PROGRAM CurrentBPUpdate
VAR
    {attribute 'pytmc' := '
        pv: @(PREFIX)K:Rate
        link: IOC:BSY0:MP01:BYKIKS_RATE
        field: EGU RateEnum
    '}
    fbBYKIK_Rate : FB_LREALFromEPICS := (
        iMaximumValidSeverity := 2);


    {attribute 'pytmc' := '
        pv: @(PREFIX)
    '}
    fbEPICS_KRate : FB_RateFromEPICS;

    {attribute 'pytmc' := '
        pv: @(PREFIX)L:BC
        link: SIOC:SYS0:MP03:SC_SXR_BC
        field: EGU BCEnum
    '}
    fbMPS_BeamClass : FB_LREALFromEPICS := (
        iMaximumValidSeverity := 2);

        {attribute 'pytmc' := '
        pv: @(PREFIX)
    '}
    fbEPICSKBeamClass : FB_BeamClassFromEPICS;

    {attribute 'pytmc' := '
        pv: @(PREFIX)K:Mode
        link: SIOC:FEES:MP01:FACMODE_RBV
    '}
    fbSXR_MachineMode : FB_LREALFromEPICS := (
        iMaximumValidSeverity := 2);

    {attribute 'pytmc' := '
        pv: @(PREFIX)
    '}
    fbEPICSLMachineMode : FB_MachineModeFromEPICS;

    {attribute 'pytmc' := '
        pv: @(PREFIX)PE
    '}
    fbKPhotonEnergy : FB_KPhotonEnergy;

    // Photon energy for the masses
    {attribute 'TcLinkTo' := 'TIIB[plc-kfe-gatt]^IO Outputs^rPhotonEnergy'}
    {attribute 'TcLinkTo' := 'TIIB[plc-rix-mot]^IO Outputs^rPhotonEnergy'}
    {attribute 'TcLinkTo' := 'TIIB[plc-rix-optics]^IO Outputs^rPhotonEnergy'}
    q_rPhotonEnergy AT %Q* : REAL;


    // Stoppers

    {attribute 'TcLinkTo' := '
                .i_StopperInLS:=TIIB[PPS Stoppers 1]^Channel 1^ST3K4 IN;
                .i_StopperOutLS:=TIIB[PPS Stoppers 1]^Channel 2^ST3K4 OUT;
                .q_StopperIN_Relay:=TIIB[PMPS_Premp]^Channel 12^ST3K4 RELAY IN;
                                '}
    st3k4Watcher : FB_KStopper(
        PMPS.K_Stopper.ST3K4,
        'ST3K4');

   {attribute 'TcLinkTo' := '
                .i_StopperInLS:=TIIB[PPS Stoppers 1]^Channel 3^ST1K2 IN;
                .i_StopperOutLS:=TIIB[PPS Stoppers 1]^Channel 4^ST1K2 OUT;
                .q_StopperIN_Relay:=TIIB[PMPS_Premp]^Channel 14^ST1K2 RELAY IN;
                                '}
    st1k2Watcher : FB_KStopper(
        PMPS.K_Stopper.ST1K2,
        'ST1K2');

    {attribute 'TcLinkTo' := '
                .i_StopperInLS:=TIIB[PPS Stoppers 1]^Channel 5^ST1K3 IN;
                .i_StopperOutLS:=TIIB[PPS Stoppers 1]^Channel 6^ST1K3 OUT;
                .q_StopperIN_Relay:=TIIB[PMPS_Premp]^Channel 7^ST1K3 RELAY IN;
                                '}
    st1k3Watcher : FB_KStopper(
        PMPS.K_Stopper.ST1K3,
        'ST1K3');

    // MR1K1 Veto
    ////////////////////////
          {attribute 'TcLinkTo' := 'TIIB[plc-rix-optics]^IO Inputs^MR1K1_Y_ENC'}
        i_MR1K1_ENC AT %I* : UDINT; // MR1K1 encoder from the rix optics system
        cMR1K1_IN_UpperLimit : UDINT := 33411000;
        cMR1K1_IN_LowerLimit : UDINT := 31911000;
        cMR1K1_OUT_UpperLimit : UDINT := 14173400;
        {attribute 'TcLinkTo' := 'TIIB[PMPS_Premp]^Channel 13^MR1K1 IN'}
        q_MR1K1_VETO AT %Q* : BOOL; // Signal to accel. MPS that MR1K1 is in
        fbMR1K1VetoDevice : FB_KVetoDevice(
            eVetoDeviceIN := K_Stopper.MR1K1_IN,
            eVetoDeviceOUT := K_Stopper.MR1K1_OUT,
            sVetoDeviceName := 'MR1K1');




    // ST4K4 Photon Terminator Veto
    {attribute 'TcLinkTo' := '
                .i_StopperInLS:=TIIB[plc-tmo-mot]^IO Inputs^bST4K4_IN;
                .i_StopperOutLS:=TIIB[plc-tmo-mot]^IO Inputs^bST4K4_OUT;
     '}
    st4k4Watcher : FB_KStopper(
        PMPS.K_Stopper.ST4K4,
        'ST4K4');


     // MR1K3 Veto
    ////////////////////////
          {attribute 'TcLinkTo' := 'TIIB[plc-txi-optics]^IO Inputs^MR1K3_Y_ENC'}
        i_MR1K3_ENC AT %I* : ULINT; // MR1K3 encoder from the txi k optics optics system
        cMR1K3_IN_UpperLimit : UDINT := 108500000 + 10000000;
        cMR1K3_IN_LowerLimit : UDINT := 108500000 - 10000000 ;
        cMR1K3_OUT_UpperLimit : UDINT := 8900000 + 100000;

        q_MR1K3_VETO AT %Q* : BOOL; // Signal to accel. MPS that MR1K3 is in
        fbMR1K3VetoDevice : FB_KVetoDevice(
            eVetoDeviceIN := K_Stopper.MR1K3_IN,
            eVetoDeviceOUT := K_Stopper.MR1K3_OUT,
            sVetoDeviceName := 'MR1K3');

    // MR2K3 Veto
    ////////////////////////
          {attribute 'TcLinkTo' := 'TIIB[plc-txi-optics]^IO Inputs^MR2K3_Y_ENC'}
        i_MR2K3_ENC AT %I* : ULINT; // MR2K3 encoder from the txi k optics system
        cMR2K3_IN_UpperLimit : UDINT := 105650000 + 10000000;
        cMR2K3_IN_LowerLimit : UDINT := 105650000 - 10000000 ;
        cMR2K3_OUT_UpperLimit : UDINT := 10000000;

        q_MR2K3_VETO AT %Q* : BOOL; // Signal to accel. MPS that MR2K3 is in
        fbMR2K3VetoDevice : FB_KVetoDevice(
            eVetoDeviceIN := K_Stopper.MR2K3_IN,
            eVetoDeviceOUT := K_Stopper.MR2K3_OUT,
            sVetoDeviceName := 'MR2K3');


    // ST1K4Veto
    // ST1K4 Test Photon stopper Veto in the FEE right before ST3K4 stopper
    st1k4Watcher :   FB_KVetoDevice(
            eVetoDeviceIN := K_Stopper.ST1K4,
            eVetoDeviceOUT := K_Stopper.DEFAULT, // not used there is no ST1K4 OUT Just a place holder
            sVetoDeviceName := 'ST1K4');
    ////////////////////////

          {attribute 'TcLinkTo' := 'TIIB[plc-kfe-motion]^IO Inputs^ST1K4_Y_ENC'}
        ST1K4_Y_ENC AT %I* : UDINT; // MR2K3 encoder from the  system
        ST1K4_IN_UpperLimit : UDINT := 4293998998 + 10000;
        ST1K4_IN_LowerLimit : UDINT := 4293998000;
        ST1K4_OUT_UpperLimit : UDINT := 8900000;

END_VAR

// Acquiring K-line rate
fbEPICS_KRate(BP:=PMPS_GVL.stCurrentBeamParameters, fbBYKIK_Rate:=fbBYKIK_Rate, FFO:=GVL.g_FastFaultOutput1);

// Acquiring photon energy
fbKPhotonEnergy(BP:=PMPS_GVL.stCurrentBeamParameters);

q_rPhotonEnergy := LREAL_TO_REAL(fbKPhotonEnergy.fbSXU.fCurrentPhotonEnergy);

//Update current photon energy
PMPS_GVL.stCurrentBeamParameters.neV := LREAL_TO_REAL(fbKPhotonEnergy.fbSXU.fCurrentPhotonEnergy);
// Acquiring K-line BeamClass
fbEPICSKBeamClass(BP:=PMPS_GVL.stCurrentBeamParameters, fbMPS_BeamClass:=fbMPS_BeamClass, FFO:=GVL.g_FastFaultOutput1);

// Acquiring K-line Machine Mode
fbEPICSLMachineMode(BP:=PMPS_GVL.stCurrentBeamParameters, fbMPS_MachineMode:=fbSXR_MachineMode, FFO:=GVL.g_FastFaultOutput1);


// Stopper readbacks
st3k4Watcher(stCurrentBP:=PMPS_GVL.stCurrentBeamParameters);
st1k2Watcher(stCurrentBP:=PMPS_GVL.stCurrentBeamParameters);
st1k3Watcher(stCurrentBP:=PMPS_GVL.stCurrentBeamParameters);
// ST4K4 Photon Terminator Veto
st4k4Watcher(stCurrentBP:=PMPS_GVL.stCurrentBeamParameters);
// MR1K1 Veto
////////////////////////
    fbMR1K1VetoDevice(
        i_bIn := cMR1K1_IN_LowerLimit < i_MR1K1_ENC	AND i_MR1K1_ENC < cMR1K1_IN_UpperLimit,
        i_bOut := i_MR1K1_ENC < cMR1K1_OUT_UpperLimit,
        q_bIN => q_MR1K1_VETO,
        stCurrentBP:= PMPS_GVL.stCurrentBeamParameters);

////////////////////////
    fbMR1K3VetoDevice(
        i_bIn := cMR1K3_IN_LowerLimit < i_MR1K3_ENC	AND i_MR1K3_ENC < cMR1K3_IN_UpperLimit,
        i_bOut := i_MR1K3_ENC < cMR1K3_OUT_UpperLimit,
        q_bIN => q_MR1K3_VETO,
        stCurrentBP:= PMPS_GVL.stCurrentBeamParameters);


// MR2K3 Veto
////////////////////////
    fbMR2K3VetoDevice(
        i_bIn := cMR2K3_IN_LowerLimit < i_MR2K3_ENC	AND i_MR2K3_ENC < cMR2K3_IN_UpperLimit,
        i_bOut := i_MR2K3_ENC < cMR2K3_OUT_UpperLimit,
        q_bIN => q_MR2K3_VETO,
        stCurrentBP:= PMPS_GVL.stCurrentBeamParameters);


// ST1K4 Photon Test stopper Veto
st1k4Watcher(i_bIn := ST1K4_IN_LowerLimit < ST1K4_Y_ENC	AND ST1K4_Y_ENC < ST1K4_IN_UpperLimit,
        i_bOut := ST1K4_Y_ENC <  ST1K4_OUT_UpperLimit,
        q_bIN => ,
        stCurrentBP:= PMPS_GVL.stCurrentBeamParameters);

END_PROGRAM

(* stored: Version 1.1.0.1, ProductVersion 3.1.4022.18
   POU CurrentBPUpdate: Id {8b324aa8-068c-4257-be00-af3f86b96ed0}, SpecialFunc None *)
